(* Schneider Machine Expert - Basic project Group 1_Automatic 2 parts assembler, file version 2.7.0.0 *)
(* ProjectInformations: Name=New project *)

HARDWARE
  Cpu 0: TM221CE16R
  EthernetConfiguration: NetworkName=M221, IpAllocationMode=FixedAddress, IpAddress=0.0.0.0, SubnetMask=0.0.0.0
  SerialLineConfiguration: Baud=Baud19200, Parity=ParityEven, DataBits=DataBits8, StopBits=StopBits1, PhysicalMedium=PhysicalMediumRs485, TransmissionMode=TransmissionModeModbusRtu, SlaveId=1, Addressing=SlaveAddressing
  MastTask: UsePeriodScanMode=false, PeriodScan=100
  FastTask: Period=255
  CpuBehavior: StartingMode=StartAsPreviousState, AutoSaveRamOnEeprom=true, WatchdogPeriod=250

SYMBOLS  (address, symbol, comment, settings)
  %M0       MOVING_X
  %M1       MOVING_Z
  %M2       ITEM_DETECTED
  %M3       LID_AT_PLACE
  %M4       LID_CLAMPED
  %M6       BASE_AT_PLACE
  %M7       BASE_CLAMPED
  %M8       BASE_POST_AT_LIMIT
  %M9       PART_LEAVING
  %M10      STARTS
  %M11      RESET
  %M12      STOPS
  %M16      MOVE_X
  %M17      MOVE_Z
  %M18      GRAB
  %M19      LIDS_CONVEYOR
  %M20      CLAMP_LID
  %M22      BASE_CONVEYOR
  %M23      CLAMP_BASE
  %M24      BASE_POST_RAISE
  %M25      START_LIGHT
  %M27      STOP_LIGHT
  %M28      PROCESS_1
  %M29      PROCESS_2
  %M30      PROCESS_3
  %M31      PROCESS_4
  %M32      TO_PROCESS_5
  %M33      PROCESS_5
  %M34      TO_PROCESS_6
  %M35      PROCESS_6
  %M36      PROCESS_7
  %M37      PROCESS_8
  %M38      PROCESS_9
  %M39      TO_PROCESS_10
  %M40      PROCESS_10
  %M41      PROCESS_11
  %M42      PROCESS_1A
  %M43      PROCESS_2A
  %M44      PROCESS_3A
  %M45      PROCESS_12
  %M46      PROCESS_13
  %M47      PROCESS_14
  %M48      PROCESS_15
  %M49      PROCESS_16
  %TM0      TIME  [Preset=1, Base=OneSecond]
  %TM1      TIME_2  [Preset=1, Base=OneSecond]
  %TM2      TIME_3  [Preset=1, Base=OneSecond]
  %Q0.0     PROSES_1
  %Q0.1     PROSES_2

POU New POU
  (* SectionNumber=1 *)

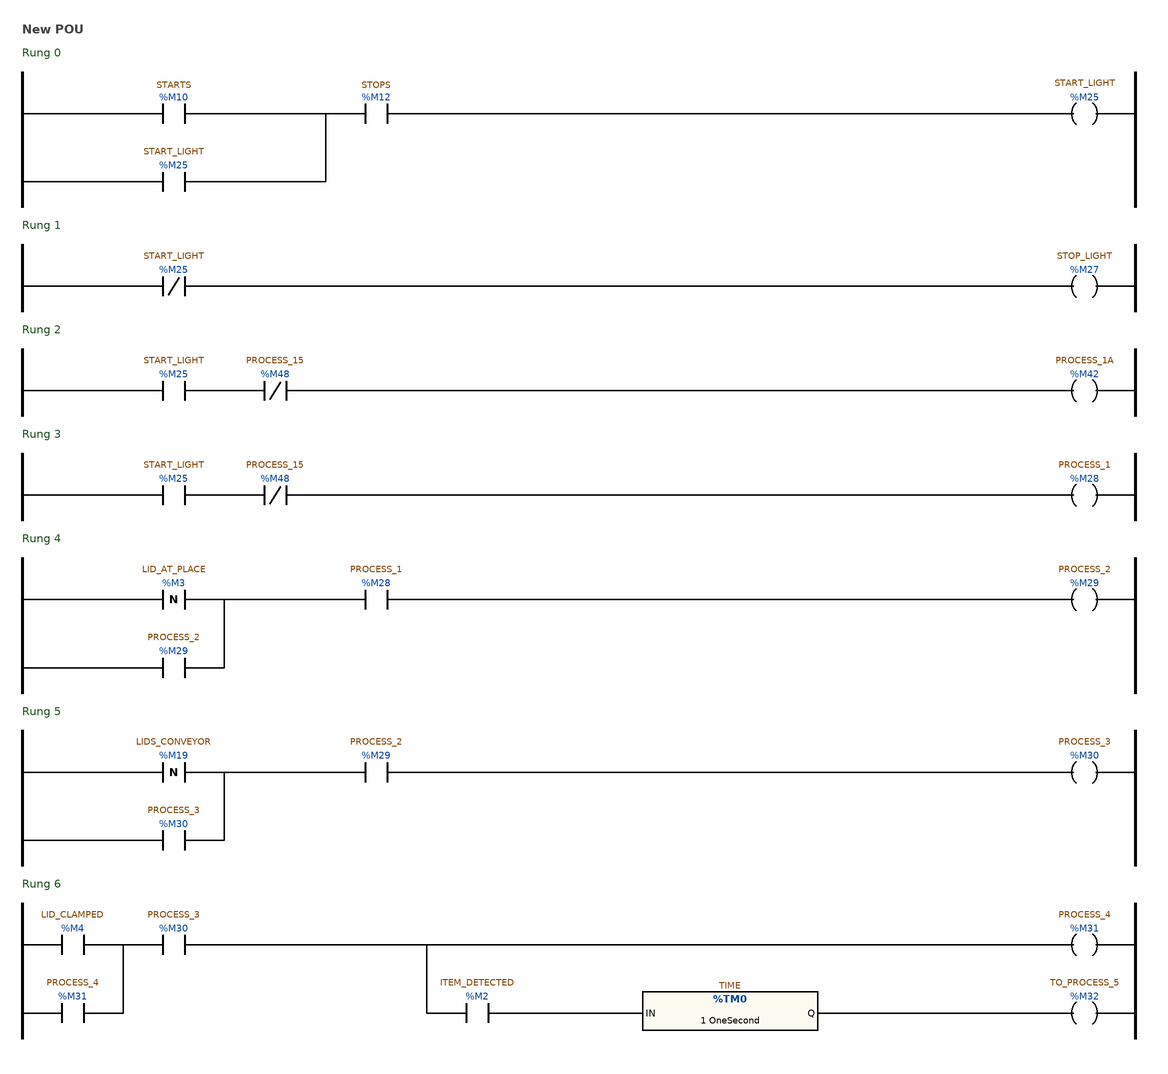

// Rung 0
  LD %M10                 (* STARTS *)
  OR %M25                 (* START_LIGHT *)
  AND %M12                (* STOPS *)
  ST %M25                 (* START_LIGHT *)
  // as ST:
  //   START_LIGHT := (STARTS OR START_LIGHT) AND STOPS;

// Rung 1
  LDN %M25                (* START_LIGHT *)
  ST %M27                 (* STOP_LIGHT *)
  // as ST:
  //   STOP_LIGHT := NOT START_LIGHT;

// Rung 2
  LD %M25                 (* START_LIGHT *)
  ANDN %M48               (* PROCESS_15 *)
  ST %M42                 (* PROCESS_1A *)
  // as ST:
  //   PROCESS_1A := START_LIGHT AND NOT PROCESS_15;

// Rung 3
  LD %M25                 (* START_LIGHT *)
  ANDN %M48               (* PROCESS_15 *)
  ST %M28                 (* PROCESS_1 *)
  // as ST:
  //   PROCESS_1 := START_LIGHT AND NOT PROCESS_15;

// Rung 4
  LDF %M3                 (* LID_AT_PLACE *)
  OR %M29                 (* PROCESS_2 *)
  AND %M28                (* PROCESS_1 *)
  ST %M29                 (* PROCESS_2 *)
  // as ST:
  //   PROCESS_2 := (FALLING(LID_AT_PLACE) OR PROCESS_2) AND PROCESS_1;

// Rung 5
  LDF %M19                (* LIDS_CONVEYOR *)
  OR %M30                 (* PROCESS_3 *)
  AND %M29                (* PROCESS_2 *)
  ST %M30                 (* PROCESS_3 *)
  // as ST:
  //   PROCESS_3 := (FALLING(LIDS_CONVEYOR) OR PROCESS_3) AND PROCESS_2;

// Rung 6
  LD 1
  MULTIFB
  LD 1
  AND %M4                 (* LID_CLAMPED *)
  OR %M31                 (* PROCESS_4 *)
  AND %M30                (* PROCESS_3 *)
  ST %MW2009:X0
  LD %MW2009:X0
  ST %M31                 (* PROCESS_4 *)
  BLK %TM0                (* TIME *)
  LD %MW2009:X0
  AND %M2                 (* ITEM_DETECTED *)
  IN
  OUT_BLK
  LD Q
  ST %M32                 (* TO_PROCESS_5 *)
  END_BLK
  MULTIFB
  // as ST:
  //   _t1 := (LID_CLAMPED OR PROCESS_4) AND PROCESS_3;
  //   PROCESS_4 := _t1;
  //   TIME(IN := _t1 AND ITEM_DETECTED);
  //   TO_PROCESS_5 := TIME.Q;

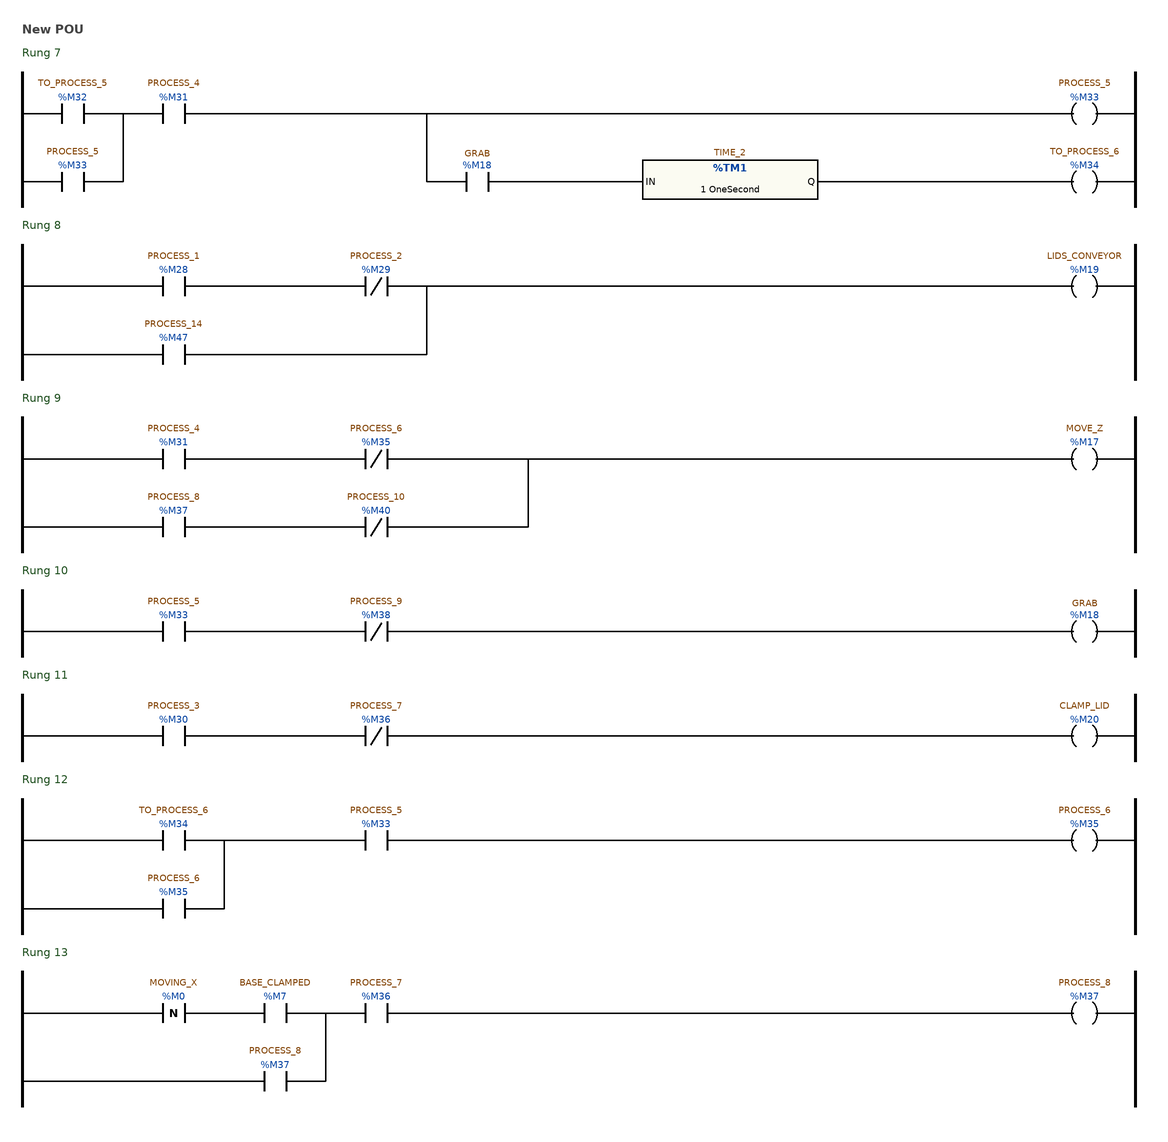

// Rung 7
  LD 1
  MULTIFB
  LD 1
  AND %M32                (* TO_PROCESS_5 *)
  OR %M33                 (* PROCESS_5 *)
  AND %M31                (* PROCESS_4 *)
  ST %MW2009:X0
  LD %MW2009:X0
  ST %M33                 (* PROCESS_5 *)
  BLK %TM1                (* TIME_2 *)
  LD %MW2009:X0
  AND %M18                (* GRAB *)
  IN
  OUT_BLK
  LD Q
  ST %M34                 (* TO_PROCESS_6 *)
  END_BLK
  MULTIFB
  // as ST:
  //   _t1 := (TO_PROCESS_5 OR PROCESS_5) AND PROCESS_4;
  //   PROCESS_5 := _t1;
  //   TIME_2(IN := _t1 AND GRAB);
  //   TO_PROCESS_6 := TIME_2.Q;

// Rung 8
  LD %M28                 (* PROCESS_1 *)
  ANDN %M29               (* PROCESS_2 *)
  OR %M47                 (* PROCESS_14 *)
  ST %M19                 (* LIDS_CONVEYOR *)
  // as ST:
  //   LIDS_CONVEYOR := PROCESS_1 AND NOT PROCESS_2 OR PROCESS_14;

// Rung 9
  LD %M31                 (* PROCESS_4 *)
  ANDN %M35               (* PROCESS_6 *)
  OR( %M37                (* PROCESS_8 *)
  ANDN %M40               (* PROCESS_10 *)
  )
  ST %M17                 (* MOVE_Z *)
  // as ST:
  //   MOVE_Z := PROCESS_4 AND NOT PROCESS_6 OR PROCESS_8 AND NOT PROCESS_10;

// Rung 10
  LD %M33                 (* PROCESS_5 *)
  ANDN %M38               (* PROCESS_9 *)
  ST %M18                 (* GRAB *)
  // as ST:
  //   GRAB := PROCESS_5 AND NOT PROCESS_9;

// Rung 11
  LD %M30                 (* PROCESS_3 *)
  ANDN %M36               (* PROCESS_7 *)
  ST %M20                 (* CLAMP_LID *)
  // as ST:
  //   CLAMP_LID := PROCESS_3 AND NOT PROCESS_7;

// Rung 12
  LD %M34                 (* TO_PROCESS_6 *)
  OR %M35                 (* PROCESS_6 *)
  AND %M33                (* PROCESS_5 *)
  ST %M35                 (* PROCESS_6 *)
  // as ST:
  //   PROCESS_6 := (TO_PROCESS_6 OR PROCESS_6) AND PROCESS_5;

// Rung 13
  LDF %M0                 (* MOVING_X *)
  AND %M7                 (* BASE_CLAMPED *)
  OR %M37                 (* PROCESS_8 *)
  AND %M36                (* PROCESS_7 *)
  ST %M37                 (* PROCESS_8 *)
  // as ST:
  //   PROCESS_8 := (FALLING(MOVING_X) AND BASE_CLAMPED OR PROCESS_8) AND PROCESS_7;

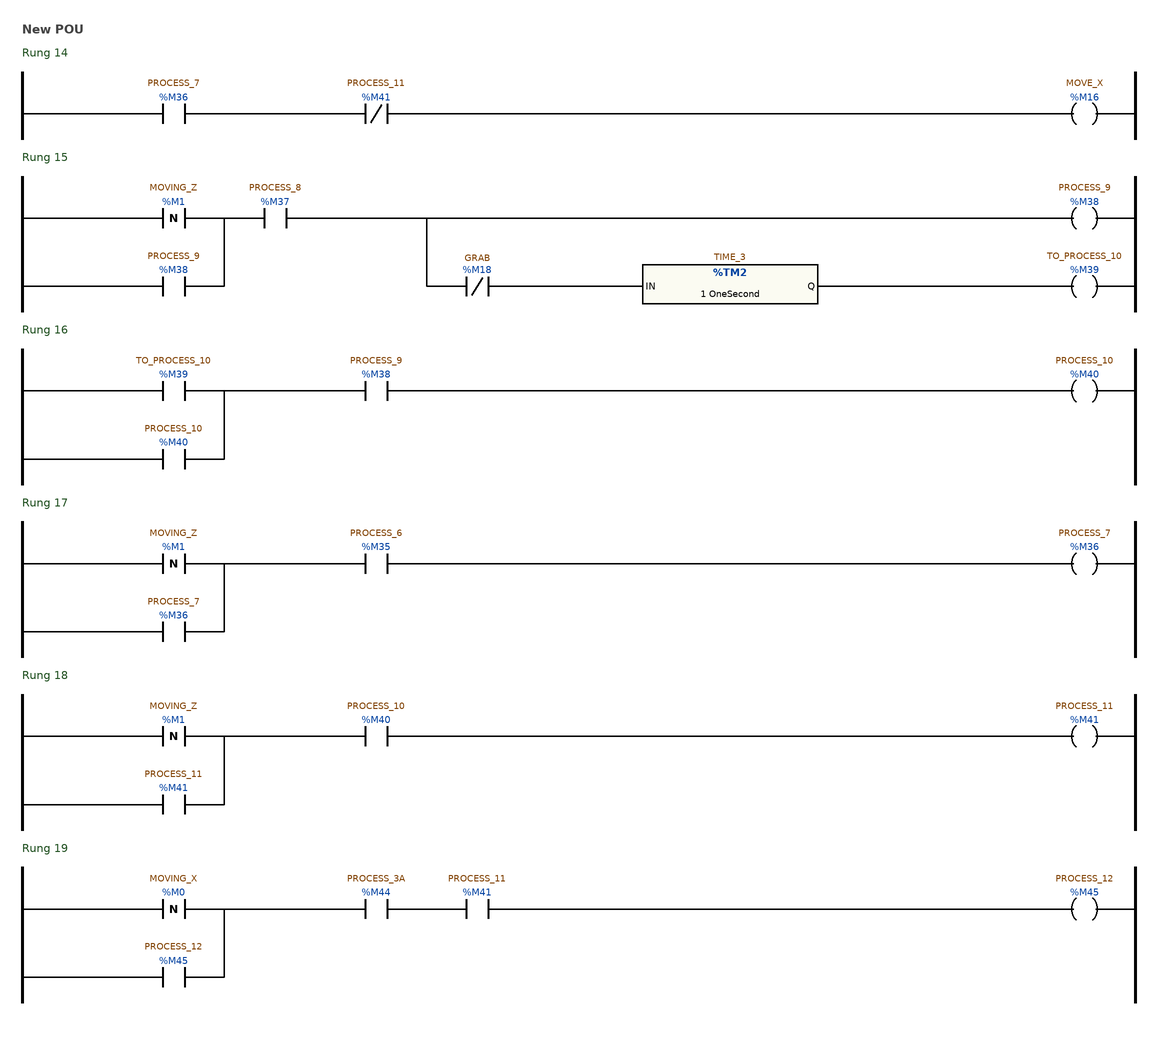

// Rung 14
  LD %M36                 (* PROCESS_7 *)
  ANDN %M41               (* PROCESS_11 *)
  ST %M16                 (* MOVE_X *)
  // as ST:
  //   MOVE_X := PROCESS_7 AND NOT PROCESS_11;

// Rung 15
  LD 1
  MULTIFB
  LD 1
  ANDF %M1                (* MOVING_Z *)
  OR %M38                 (* PROCESS_9 *)
  AND %M37                (* PROCESS_8 *)
  ST %MW2009:X0
  LD %MW2009:X0
  ST %M38                 (* PROCESS_9 *)
  BLK %TM2                (* TIME_3 *)
  LD %MW2009:X0
  ANDN %M18               (* GRAB *)
  IN
  OUT_BLK
  LD Q
  ST %M39                 (* TO_PROCESS_10 *)
  END_BLK
  MULTIFB
  // as ST:
  //   _t1 := (FALLING(MOVING_Z) OR PROCESS_9) AND PROCESS_8;
  //   PROCESS_9 := _t1;
  //   TIME_3(IN := _t1 AND NOT GRAB);
  //   TO_PROCESS_10 := TIME_3.Q;

// Rung 16
  LD %M39                 (* TO_PROCESS_10 *)
  OR %M40                 (* PROCESS_10 *)
  AND %M38                (* PROCESS_9 *)
  ST %M40                 (* PROCESS_10 *)
  // as ST:
  //   PROCESS_10 := (TO_PROCESS_10 OR PROCESS_10) AND PROCESS_9;

// Rung 17
  LDF %M1                 (* MOVING_Z *)
  OR %M36                 (* PROCESS_7 *)
  AND %M35                (* PROCESS_6 *)
  ST %M36                 (* PROCESS_7 *)
  // as ST:
  //   PROCESS_7 := (FALLING(MOVING_Z) OR PROCESS_7) AND PROCESS_6;

// Rung 18
  LDF %M1                 (* MOVING_Z *)
  OR %M41                 (* PROCESS_11 *)
  AND %M40                (* PROCESS_10 *)
  ST %M41                 (* PROCESS_11 *)
  // as ST:
  //   PROCESS_11 := (FALLING(MOVING_Z) OR PROCESS_11) AND PROCESS_10;

// Rung 19
  LDF %M0                 (* MOVING_X *)
  OR %M45                 (* PROCESS_12 *)
  AND %M44                (* PROCESS_3A *)
  AND %M41                (* PROCESS_11 *)
  ST %M45                 (* PROCESS_12 *)
  // as ST:
  //   PROCESS_12 := (FALLING(MOVING_X) OR PROCESS_12) AND PROCESS_3A AND PROCESS_11;

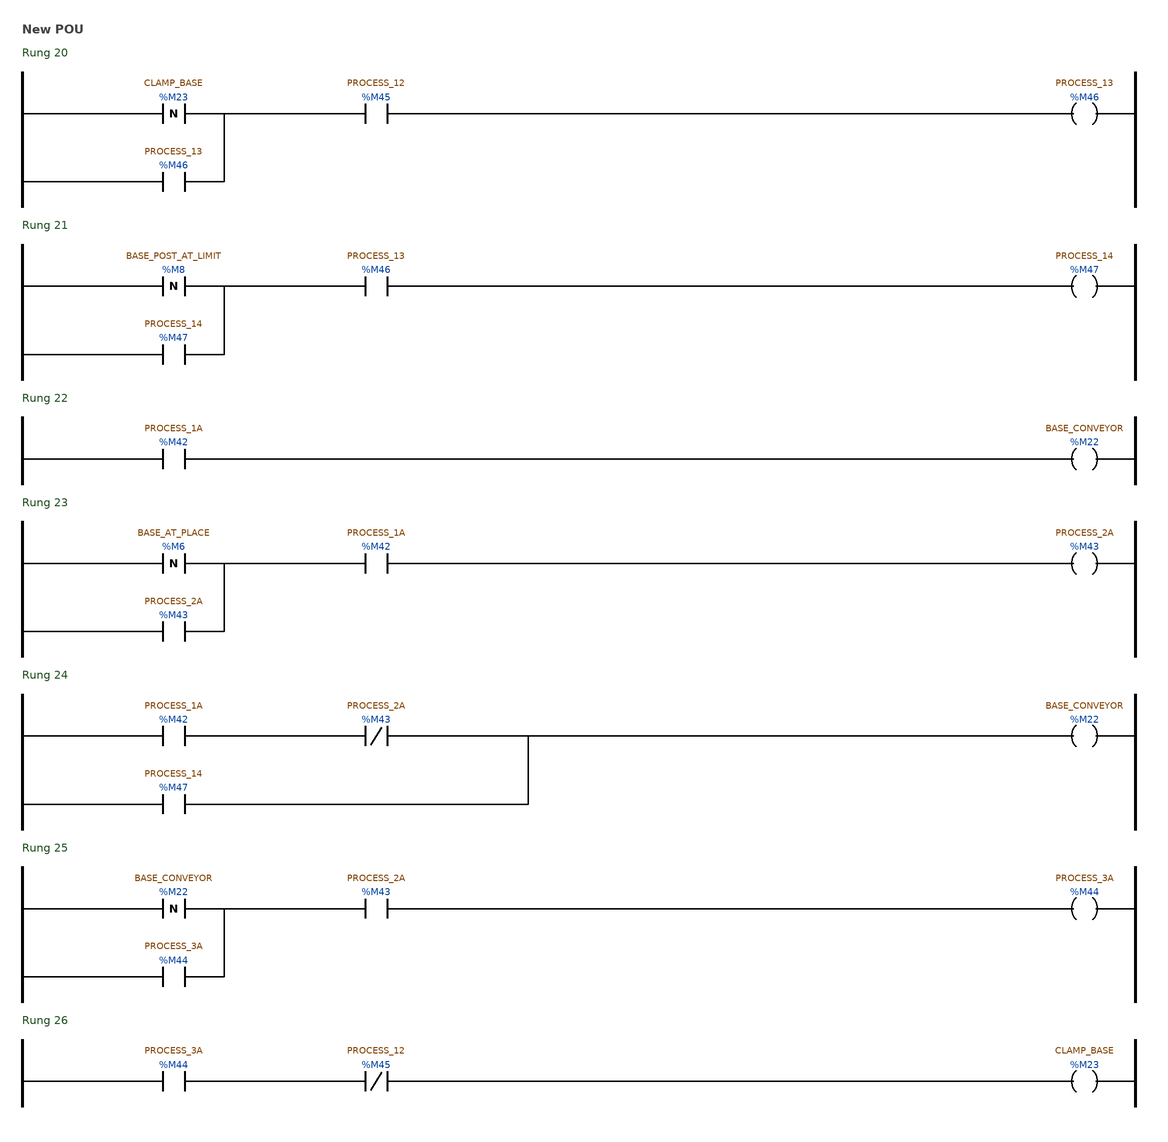

// Rung 20
  LDF %M23                (* CLAMP_BASE *)
  OR %M46                 (* PROCESS_13 *)
  AND %M45                (* PROCESS_12 *)
  ST %M46                 (* PROCESS_13 *)
  // as ST:
  //   PROCESS_13 := (FALLING(CLAMP_BASE) OR PROCESS_13) AND PROCESS_12;

// Rung 21
  LDF %M8                 (* BASE_POST_AT_LIMIT *)
  OR %M47                 (* PROCESS_14 *)
  AND %M46                (* PROCESS_13 *)
  ST %M47                 (* PROCESS_14 *)
  // as ST:
  //   PROCESS_14 := (FALLING(BASE_POST_AT_LIMIT) OR PROCESS_14) AND PROCESS_13;

// Rung 22
  LD %M42                 (* PROCESS_1A *)
  ST %M22                 (* BASE_CONVEYOR *)
  // as ST:
  //   BASE_CONVEYOR := PROCESS_1A;

// Rung 23
  LDF %M6                 (* BASE_AT_PLACE *)
  OR %M43                 (* PROCESS_2A *)
  AND %M42                (* PROCESS_1A *)
  ST %M43                 (* PROCESS_2A *)
  // as ST:
  //   PROCESS_2A := (FALLING(BASE_AT_PLACE) OR PROCESS_2A) AND PROCESS_1A;

// Rung 24
  LD %M42                 (* PROCESS_1A *)
  ANDN %M43               (* PROCESS_2A *)
  OR %M47                 (* PROCESS_14 *)
  ST %M22                 (* BASE_CONVEYOR *)
  // as ST:
  //   BASE_CONVEYOR := PROCESS_1A AND NOT PROCESS_2A OR PROCESS_14;

// Rung 25
  LDF %M22                (* BASE_CONVEYOR *)
  OR %M44                 (* PROCESS_3A *)
  AND %M43                (* PROCESS_2A *)
  ST %M44                 (* PROCESS_3A *)
  // as ST:
  //   PROCESS_3A := (FALLING(BASE_CONVEYOR) OR PROCESS_3A) AND PROCESS_2A;

// Rung 26
  LD %M44                 (* PROCESS_3A *)
  ANDN %M45               (* PROCESS_12 *)
  ST %M23                 (* CLAMP_BASE *)
  // as ST:
  //   CLAMP_BASE := PROCESS_3A AND NOT PROCESS_12;

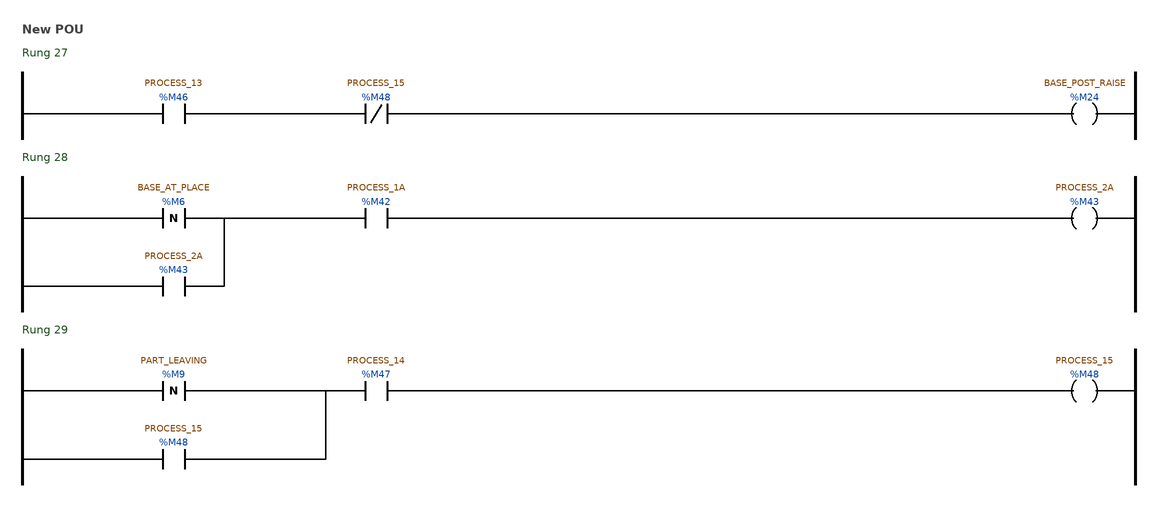

// Rung 27
  LD %M46                 (* PROCESS_13 *)
  ANDN %M48               (* PROCESS_15 *)
  ST %M24                 (* BASE_POST_RAISE *)
  // as ST:
  //   BASE_POST_RAISE := PROCESS_13 AND NOT PROCESS_15;

// Rung 28
  LDF %M6                 (* BASE_AT_PLACE *)
  OR %M43                 (* PROCESS_2A *)
  AND %M42                (* PROCESS_1A *)
  ST %M43                 (* PROCESS_2A *)
  // as ST:
  //   PROCESS_2A := (FALLING(BASE_AT_PLACE) OR PROCESS_2A) AND PROCESS_1A;

// Rung 29
  LDF %M9                 (* PART_LEAVING *)
  OR %M48                 (* PROCESS_15 *)
  AND %M47                (* PROCESS_14 *)
  ST %M48                 (* PROCESS_15 *)
  // as ST:
  //   PROCESS_15 := (FALLING(PART_LEAVING) OR PROCESS_15) AND PROCESS_14;
